// TwinCAT 3 PLC project Untitled1
// ProgramVersion: 3.1.4023.0
// libraries:
//   Tc2_Standard, * (Beckhoff Automation GmbH)
//   Tc2_System, * (Beckhoff Automation GmbH)
//   Tc3_Module, * (Beckhoff Automation GmbH)
// project tree:
//   / GlobalTextList.TcGTLO, PlcTask.TcTTO, Visualization Manager.TcVMO (not stored)
//   POUs/ MAIN.TcPOU, FB_MalzemeSecme.TcPOU
//   VISUs/ VISU_1.TcVIS
// real-time tasks:
//   TASK PlcTask: cycle T#10ms, priority 20, ADS port 350

CONFIGURATION Untitled1
    RESOURCE PLC ON TwinCAT3
        TASK PlcTask(INTERVAL := T#10ms, PRIORITY := 20);
        PROGRAM MAIN WITH PlcTask : MAIN;
    END_RESOURCE
END_CONFIGURATION

// ---- POUs/MAIN.TcPOU
PROGRAM MAIN
VAR
	nState: INT;
	bButon: BOOL;
	bSensor1: BOOL;
	ftrig1: F_TRIG;
	bHat: BOOL;
	rtrig1: R_TRIG;
	bSensor2: BOOL;
	random1: DRAND;
	nYukseklik: INT;
	Select1: FB_MalzemeSecme;
	T1: TON;
	T2: TON;
	T3: TON;
	bKol1: BOOL;
	bKutuSens1: BOOL;
	bKutuSens2: BOOL;
	bKutuSens3: BOOL;
	rtrig2: R_TRIG;
	rtrig3: R_TRIG;
	rtrig4: R_TRIG;
	bKol2: BOOL;
	bKol3: BOOL;
	nKisaKutu: INT;
	nOrtaKutu: INT;
	nUzunKutu: INT;
	sInfoMsg: STRING;
	sMsgKisa_1: STRING(255);
	sMsgOrta_1: STRING(255);
	sMsgUzun_1: STRING(255);
	sMsgYukseklik: STRING(255);
END_VAR


ACT_PRG();

ACT_VisuMsg();

ACTION ACT_PRG:

ftrig1(CLK:= bSensor1 , Q=> );

rtrig1(CLK:= bSensor2 , Q=> );


rtrig2(CLK:= bKutuSens1 , Q=> ); // Kısa malzeme kutusu sensörü

rtrig3(CLK:= bKutuSens2 , Q=> ); // Orta malzeme kutusu sensörü

rtrig4(CLK:= bKutuSens3 , Q=> ); // Uzun malzeme kutusu sensörü


CASE nState OF 
	

	0:
	
	IF bButon THEN 
		
		nState := 10;
		
	END_IF
	
	
	10:
	
	sInfoMsg := 'Malzeme Bekleniyor.';
	
	IF ftrig1.Q THEN
		
		nState := 20;
		
	END_IF
	
	
	20:
	
	bHat := TRUE;
	
	sInfoMsg := 'Hat Aktif, Malzemenin Konuma Gelmesi Bekleniyor.';

	IF rtrig1.Q THEN
		
		bHat := FALSE;
		
		random1(Seed:=10 , Num=> );
		nYukseklik := LREAL_TO_INT(random1.Num * 100);
		
		nState := 30;
		
	END_IF
	
	
	30:
		
	Select1(nValue:=nYukseklik,
			nStateOut=>nState, 
			sMsg =>sInfoMsg );	
	
	
	32:
	
		bHat := TRUE;
		T1(IN:=TRUE , PT:=T#2S);
		
		IF T1.Q THEN
			nState := 42;
			T1(IN:=FALSE);
			bHat := FALSE;
		END_IF
	
	34:
	
		bHat := TRUE;
		T2(IN:=TRUE , PT:=T#4S);
		
		IF T2.Q THEN
			nState := 44;
			T2(IN:=FALSE);
			bHat := FALSE;
		END_IF
	
	
	36:
		bHat := TRUE;
		T3(IN:=TRUE , PT:=T#6S);
		
		IF T3.Q THEN
			nState := 46;
			T3(IN:=FALSE);
			bHat := FALSE;
		END_IF
		
		
	42:
		
		bKol1 := TRUE;
		sInfoMsg	:=	'Kısa Boyutlu Malzeme Kutusuna Koyuluyor.';
		
		IF rtrig2.Q THEN
			
			bKol1 := FALSE;
			
			nKisaKutu := nKisakutu + 1;
			
			nState := 0;
			
		END_IF
		
		
	
	44:
	
		bKol2 := TRUE;
		sInfoMsg	:=	'Orta Boyutlu Malzeme Kutusuna Koyuluyor.';
		
		IF rtrig3.Q THEN
			
			bKol2 := FALSE;
			
			nOrtaKutu := nOrtaKutu + 1;
			
			nState := 0;
			
		END_IF	

	46:
		bKol3:= TRUE;
		sInfoMsg	:=	'Uzun Boyutlu Malzeme Kutusuna Koyuluyor.';
		
		IF rtrig4.Q THEN
			
			bKol3 := FALSE;
			
			nUzunKutu := nUzunKutu + 1;
			
			nState := 0;
			
		END_IF	
	
			
END_CASE


	IF NOT bButon THEN 
		
		nState := 0;
		sInfoMsg := 'Sistem Kapali.';
		bKol1 := FALSE;
		bKol2 := FALSE;
		bKol3 := FALSE;
		T1(IN:=FALSE);
		T2(IN:=FALSE);
		T3(IN:=FALSE);
		
	END_IF
END_ACTION

ACTION ACT_VisuMsg:


sMsgKisa_1 := CONCAT(STR1:='Kisa Malzeme Kutusunda ' , STR2:= INT_TO_STRING(nKisaKutu) );
sMsgKisa_1 := CONCAT(STR1:=sMsgKisa_1 , STR2:= ' Malzeme Var' );

sMsgOrta_1 := CONCAT(STR1:='Orta Malzeme Kutusunda ' , STR2:= INT_TO_STRING(nOrtaKutu) );
sMsgOrta_1 := CONCAT(STR1:=sMsgOrta_1 , STR2:= ' Malzeme Var' );

sMsgUzun_1 := CONCAT(STR1:='Uzun Malzeme Kutusunda ' , STR2:= INT_TO_STRING(nUzunKutu) );
sMsgUzun_1 := CONCAT(STR1:=sMsgUzun_1 , STR2:= ' Malzeme Var' );

sMsgYukseklik := CONCAT(STR1:='Malzeme Yüksekligi: ' , STR2:= INT_TO_STRING(nYukseklik) );
sMsgYukseklik := CONCAT(STR1:=sMsgYukseklik , STR2:= ' [cm]' );
END_ACTION

END_PROGRAM

// ---- POUs/FB_MalzemeSecme.TcPOU
FUNCTION_BLOCK FB_MalzemeSecme
VAR_INPUT
	nValue: INT;
END_VAR
VAR_OUTPUT
	nStateOut: INT;
	sMsg: STRING;
END_VAR
VAR
END_VAR



IF nValue >= 0 AND nValue <=40 THEN
	
	sMsg := 'Malzeme Kısa Boyutlu.';
	
	nStateOut := 32;
	
ELSIF nValue >40 AND nValue <= 70 THEN

	sMsg := 'Malzeme Orta Boyutlu.';
	nStateOut := 34;
	
ELSIF nValue > 70 AND nValue <=100 THEN
		
	sMsg := 'Malzeme Uzun Boyutlu.';
	nStateOut := 36;	
	
END_IF

END_FUNCTION_BLOCK

// ---- GlobalTextList.TcGTLO
TEXTLIST GlobalTextList
  843 = '%i'
  765 = '%s'
  107 = 'bSensor1'
  283 = 'bSensor2'
  622 = 'Konveyör'
  298 = 'Kutu Sens (K)'
  547 = 'Kutu Sensor (K)'
  545 = 'Kutu Sensor (O)'
  763 = 'Kutu Sensor (U)'
  316 = 'Kutu Sensor - 1 '
  249 = 'Kutu Sensor - 13'
  334 = 'Kutu Sensor - 2'
  953 = 'Kutu Sensor - 3'
  567 = 'Kutu Sensor1'
  566 = 'Kısa Malzeme Kutusu'
  101 = 'Orta Malzeme Kutusu'
  235 = 'Sensor - 1'
  295 = 'Sensor - 2'
  906 = 'Start'
  320 = 'Uzun Malzeme Kutusu'
  291 = 'UzunMalzeme Kutusu'
  531 = 'İtici - 1'
  323 = 'İtici - 2'
  317 = 'İtici - 3'
END_TEXTLIST

// ---- VISUs/VISU_1.TcVIS
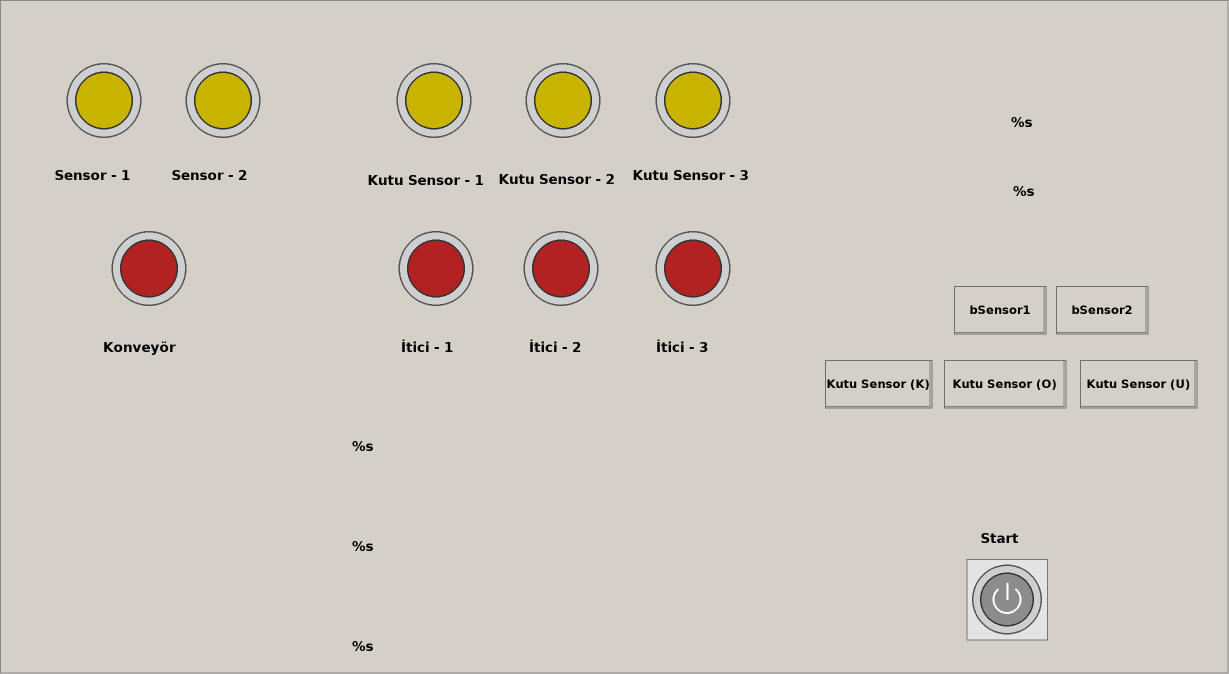
VISUALIZATION VISU_1  // 1229x674
    PowerSwitch (964,559 86x81), variable: MAIN.bButon, behaviour: TOGGLE, style: Switch-PowerSwitch-Gray
    Button (954,286 92x48), "bSensor1"
        toggle MAIN.bSensor1
    Button (1056,286 92x48), "bSensor2"
        toggle MAIN.bSensor2
    Label (951,511 97x55), "Start"
    Button (825,360 107x48), "Kutu Sensor (K)"
        toggle MAIN.bKutuSens1
    Button (944,360 122x48), "Kutu Sensor (O)"
        toggle MAIN.bKutuSens2
    Button (1080,360 117x48), "Kutu Sensor (U)"
        toggle MAIN.bKutuSens3
    Lamp1 (52,57 104x87), variable: MAIN.bSensor1, style: Lamp-Lamp1-Yellow
    Lamp1 (171,57 104x87), variable: MAIN.bSensor2, style: Lamp-Lamp1-Yellow
    Lamp1 (382,57 104x87), variable: MAIN.bKutuSens1, style: Lamp-Lamp1-Yellow
    Lamp1 (511,57 104x87), variable: MAIN.bKutuSens2, style: Lamp-Lamp1-Yellow
    Lamp1 (641,57 104x87), variable: MAIN.bKutuSens3, style: Lamp-Lamp1-Yellow
    Lamp1 (97,225 104x87), variable: MAIN.bHat, style: Lamp-Lamp1-Red
    Lamp1 (384,225 104x87), variable: MAIN.bKol1, style: Lamp-Lamp1-Red
    Lamp1 (509,225 104x87), variable: MAIN.bKol2, style: Lamp-Lamp1-Red
    Lamp1 (641,225 104x87), variable: MAIN.bKol3, style: Lamp-Lamp1-Red
    Rectangle (105,419 516x55), "%s", text variable: MAIN.sMsgKisa_1
    Rectangle (105,519 516x55), "%s", text variable: MAIN.sMsgOrta_1
    Rectangle (105,619 516x55), "%s", text variable: MAIN.sMsgUzun_1
    Label (91,320 97x55), "Konveyör"
    Label (379,320 97x55), "İtici - 1"
    Label (507,320 97x55), "İtici - 2"
    Label (634,320 97x55), "İtici - 3"
    Label (44,148 97x55), "Sensor - 1"
    Label (161,148 97x55), "Sensor - 2"
    Label (357,153 142x55), "Kutu Sensor - 1"
    Label (486,152 142x55), "Kutu Sensor - 2"
    Label (620,148 142x55), "Kutu Sensor - 3"
    Rectangle (817,95 410x55), "%s", text variable: MAIN.sInfoMsg
    Rectangle (819,164 410x55), "%s", text variable: MAIN.sMsgYukseklik
END_VISUALIZATION
